Yaskawa INFORM job: P-X(FRONIUS).JBI

/JOB
//NAME P-X(FRONIUS)
///FOLDERNAME INNE
//POS
///NPOS 9,9,9,0,0,0
///TOOL 0
///POSTYPE PULSE
///PULSE
C00000=-805,-58685,-16915,23784,70187,37121
C00001=7551,-60285,-20310,45326,70978,36888
C00002=14225,-62702,-26310,66484,71810,36398
C00003=18495,-65846,-34220,87051,73372,35738
C00004=19976,-69665,-43229,106982,76100,35225
C00005=-9612,-57992,-16692,2155,68951,37344
C00006=-17603,-58215,-19554,-19285,67278,37889
C00007=-23808,-59579,-25304,-40446,65749,38982
C00008=-27527,-61986,-32958,-61408,65146,40689
BC00000=103517,121621,531728
BC00001=103517,121620,531723
BC00002=103517,121620,531723
BC00003=103517,121620,531723
BC00004=103517,121620,531723
BC00005=103517,121620,531720
BC00006=103517,121620,531723
BC00007=103517,121620,531723
BC00008=103517,121620,531723
EC00000=0,0
EC00001=-177478,1
EC00002=-354865,1
EC00003=-532123,1
EC00004=-709909,1
EC00005=177737,0
EC00006=354971,1
EC00007=532932,1
EC00008=709881,1
//INST
///DATE 2023/10/04 15:16
///ATTR SC,RW
///GROUP1 RB1,BS1
///GROUP2 ST1
NOP
MOVJ C00000 BC00000 VJ=0.78  +MOVJ EC00000 VJ=0.78
MOVJ C00001 BC00001 VJ=0.78  +MOVJ EC00001 VJ=0.78
MOVJ C00002 BC00002 VJ=0.78  +MOVJ EC00002 VJ=0.78
MOVJ C00003 BC00003 VJ=0.78  +MOVJ EC00003 VJ=0.78
MOVJ C00004 BC00004 VJ=0.78  +MOVJ EC00004 VJ=0.78
MOVJ C00005 BC00005 VJ=0.78  +MOVJ EC00005 VJ=0.78
MOVJ C00006 BC00006 VJ=0.78  +MOVJ EC00006 VJ=0.78
MOVJ C00007 BC00007 VJ=0.78  +MOVJ EC00007 VJ=0.78
MOVJ C00008 BC00008 VJ=0.78  +MOVJ EC00008 VJ=0.78
END
